// TIA Portal V21 export
DATA_BLOCK "Percorso"   // DB9
{ S7_Optimized_Access := 'TRUE' }
// stored: MemoryReserve 100
   VAR RETAIN
      Stazione { S7_SetPoint := 'True'} : Array[0.."K_NumStazione"] of "Std_Stazione";
   END_VAR
   VAR
      Funzioni : Struct
         Inizializza : Bool := FALSE;
      END_STRUCT;
      Hmi : Struct
         CaricaInLavoro : Bool := FALSE;
         ResettaTuttoOffline : Bool := FALSE;
         RipristinaOnline : Bool := FALSE;
         CompilaVerificaConflitti : Bool := FALSE;
         AggiornaConfigurazione : Bool := FALSE;
      END_STRUCT;
   END_VAR
BEGIN
END_DATA_BLOCK
